(* IEC 61131-3 sources: conversion/src/ToHex, 2 files *)

(* ---- GetHexValueOfChar.st ---- *)
USING System.Strings;

NAMESPACE Simatic.Ax.Conversion

    // returns the hex value as byte of a hex character
    // Example 'a' --> BYTE#16#a
    // Valid characters: [A-Fa-f0-9]
    // Return vlaue: character is valid
    FUNCTION INTERNAL GetHexValueOfChar : BOOL
        VAR_INPUT
            c : CHAR;
        END_VAR
        VAR_OUTPUT
            result : BYTE;
        END_VAR
        GetHexValueOfChar := TRUE;
        CASE c OF
            '0':
                result := BYTE#16#0;
                RETURN;
            '1':
                result := BYTE#16#1;
                RETURN;
            '2':
                result := BYTE#16#2;
                RETURN;
            '3':
                result := BYTE#16#3;
                RETURN;
            '4':
                result := BYTE#16#4;
                RETURN;
            '5':
                result := BYTE#16#5;
                RETURN;
            '6':
                result := BYTE#16#6;
                RETURN;
            '7':
                result := BYTE#16#7;
                RETURN;
            '8':
                result := BYTE#16#8;
                RETURN;
            '9':
                result := BYTE#16#9;
                RETURN;
            'a', 'A':
                result := BYTE#16#A; //a A
                RETURN;
            'b', 'B':
                result := BYTE#16#B; //b B
                RETURN;
            'c', 'C':
                result := BYTE#16#C; //c C
                RETURN;
            'd', 'D':
                result := BYTE#16#D; //d D
                RETURN;
            'e', 'E':
                result := BYTE#16#E; //e E
                RETURN;
            'f', 'F':
                result := BYTE#16#F; //f F
                RETURN;
        ELSE
            // ERROR ;
            GetHexValueOfChar := FALSE;
            RETURN;
        END_CASE;
        ;
    END_FUNCTION

END_NAMESPACE

(* ---- StringToHex.st ---- *)
USING System.Strings;

NAMESPACE Simatic.Ax.Conversion.Strings

    /// This function convert a string contining a hex number into a hex number
    /// Example 'a231' --> WORD#16#a231
    /// Return values:
    /// WORD#16#0000 no error
    /// WORD#16#0007 invalid character
    /// WORD#16#8182 Input buffer is too small for data in the N parameter
    /// WORD#16#8482 Output buffer is too small for data in the N parameter
    FUNCTION ToHex : WORD
        VAR_INPUT
            str : STRING; // Pointer to ASCII character string
            n : INT; // Number of ASCII characters to be converted
        END_VAR
        VAR_OUTPUT
            result : DWORD; // Hexadecimal number
        END_VAR
        VAR_TEMP
            i : INT;
            tempCharacter : USINT;
            tempValue : BYTE;
            tempDword : DWORD;
            tempResult : DWORD;
            tempSuccess : BOOL;
        END_VAR
        // Check input length
        IF n > lengthOF(str) THEN
            ToHex := WORD#16#8182; // Input buffer is too small for data in the N parameter
            RETURN;
            ;
        END_IF;
        // Check buffer size
        IF n > 8 THEN
            ToHex := WORD#16#8482; // Output buffer is too small for data in the N parameter
            RETURN;
        END_IF;
        // Valid ASCII [0-9a-fA-F]
        FOR i := 1 TO n DO
            IF (GetHexValueOfChar(str[i], tempValue)) THEN
                tempDword := tempValue;
                tempDword := SHL(tempDword, TO_UINT((n - i) * 4));
                tempResult := tempResult OR TO_DWORD(TO_INT(tempDword));
            ELSE
                // ERROR invalid character;
                ToHex := WORD#16#0007; // Invalid charcter
                RETURN;
            END_IF;
            ;
        END_FOR;
        result := tempResult;
        ToHex := WORD#16#0000; // no Error
        ;
    END_FUNCTION

END_NAMESPACE
